// TIA Portal V19 export
TYPE "LAF_typeDevDiagGlobal"
TITLE = PN_DEV_DIAG
// This data type contains global information for the HMI Pop-up.  
// 
// **PLC Data types**  
// * [LAF_typeDevDiagNoOfDevices](../Library%20Types/LAF_typeDevDiagNoOfDevices.htm)
// Autor: SICAR
// stored: Access Published
   STRUCT
      geoAddressSystem { ExternalWritable := 'False'} : UInt;   // mittels "LOG2GEO" aus log.Adresse (Systemkonstante) die geo.Adresse des PNIO-System ermitteln / Evaluate geo address from log address
      maxDevices { ExternalWritable := 'False'} : DInt;   // Input-Abbild / Input image
      maxModuls { ExternalWritable := 'False'} : DInt;   // Input-Abbild / Input image
      lowestDevNoConfig { ExternalWritable := 'False'} : DInt;   // niedrgste PN-GeräteNr. / lowest PN device number
      highestDevNoConfig { ExternalWritable := 'False'} : DInt;   // höchste PN-GeräteNr. / highest PN device number
      numberOfDevices { ExternalWritable := 'False'} : "LAF_typeDevDiagNoOfDevices";   // Mittels"DeviceStates" ermittelte Info / Via "DevicesStates" evaluated info
      devDiagSummary { ExternalWritable := 'False'} : Bool;   // Summensignal PN-Diagnosefehler / Collective signal PN-Diagnostic error
      blockBusyAfterNewStart { ExternalWritable := 'False'} : Bool;   // FB läuft mit "Lesen von Daten", die nur einmalig nach CPU-Neustart gelesen werden. / FB busy with reading unique information after PLC startup
      manualReadAll : Bool;   // Manueller Anstoss ; erneutes Einlesen aller Daten/Infos / Manual trigger; renew informations
      resetHistoryAll : Bool;   // ResetHistoryAll von HMI / ResetHistoryAll from HMI
   END_STRUCT;
END_TYPE
